TYPE "UDT_SyncPhotocel_Hmi_V0.01"
VERSION : 0.1
   STRUCT
      tHMR { ExternalWritable := 'False'} : Struct   // {[Unit]|[Scada Unit]|[LowLimit]|[HigLimit]|[Acces]}
         xPhotocell { ExternalWritable := 'False'} : Bool;   // Photocell Present {x|x|x|x|O}
         iState { ExternalWritable := 'False'} : Int;   // State (1=No anomaly, 7=Anomaly) {x|x|x|x|O}
         dPositionX_mm { ExternalWritable := 'False'} : DInt;   // Positon Photocell {x|x|x|x|O}
         dPositionY_mm { ExternalWritable := 'False'} : DInt;   // Positon Photocell {x|x|x|x|O}
         sName { ExternalWritable := 'False'} : String;   // Name Photocell {x|x|x|x|O}
      END_STRUCT;
   END_STRUCT;

END_TYPE

DATA_BLOCK "SyncPhotocel_Hmi"
{ S7_Optimized_Access := 'FALSE' }
VERSION : 0.1
NON_RETAIN
   STRUCT
      tPhotcel : Array["STARTARRAY".."DNUMBERPHSYNC"] of "UDT_SyncPhotocel_Hmi_V0.01";
   END_STRUCT;


BEGIN

END_DATA_BLOCK

